# EPICS substitutions: ek9000App/Db/EL3001.substitutions
file EL3001.template
{       pattern
        {
                TERMINAL,

        }
        {
        }
}
